// Mitsubishi GX Works2 project: IR   PLC: FX2N/FX2NC

PROGRAM MAIN
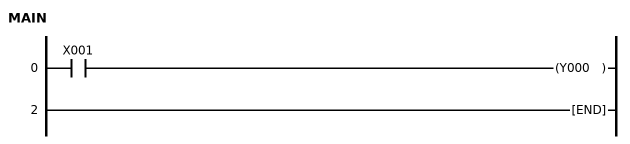
0     LD      X001
      OUT     Y000
2     END
END_PROGRAM
